Universal Robots PolyScope program: rtde_control_loop.urp

Program rtde_control_loop (installation=default directory=/programs createdIn=3.2.19275 lastSavedIn=5.13.0 robotSerialNumber=20225502595)
Calibrated DH parameters: a=[0.000032, -0.354602, -0.349314, -0.000114, 0.000079, 0]; d=[0.162572, 168.876417, -198.440969, 29.697991, 0.099792, 0.099551]; alpha=[1.570395, -0.001391, 0.006062, 1.570232, -1.569128, 0]; deltaTheta=[0, -0.584958, 0.110941, 0.474028, -0.000001, 0]
InitVariablesNode
BeforeStart
  setp := Joint_6_name
  Script: rtde_set_watchdog("input_int_register_0", 1, "PAUSE")
Robot Program (runOnlyOnce=false)
  Script: sync()
  MoveJ speed 60 deg/s, acceleration 80 deg/s^2 (useActiveTCP=true) feature=Base
    Waypoint Waypoint_1: TCP in base x=-26.855 y=-347.092 z=270.918 mm, rx=-0.0078 ry=3.1136 rz=-0.0162 rad; joints [-75.407, -74.048, -112.936, -82.13, 91.685, 14.557] deg; TCP offset x=0 y=50 z=155 mm, rx=0 ry=0 rz=0 rad
  If read_input_integer_register(1)≟1
    Script: write_output_integer_register(0, 0)
    MoveL speed 250 mm/s, acceleration 1200 mm/s^2 (useActiveTCP=true) feature=Base
      Waypoint Variable (Variable): variable=setp
    URCap qb Grasp (qbrobotics, qbrobotics®) dataModel(control_mode=deflection, grasp_command=78, grasp_threshold=100, grasp_velocity=100, grasp_stiffness=0)
    MoveJ speed 60 deg/s, acceleration 80 deg/s^2 (useActiveTCP=true) feature=Base
      Waypoint Waypoint_1: TCP in base x=-26.855 y=-347.092 z=270.918 mm, rx=-0.0078 ry=3.1136 rz=-0.0162 rad; joints [-75.407, -74.048, -112.936, -82.13, 91.685, 14.557] deg
      Waypoint Waypoint_2: TCP in base x=181.876 y=-239.045 z=110.303 mm, rx=-0.0609 ry=3.1315 rz=0.0832 rad; joints [-37.025, -75.759, -136.666, -59.157, 92.873, 51.044] deg
    URCap qb Grasp (qbrobotics, qbrobotics®) dataModel(control_mode=position, grasp_stiffness=50, grasp_command=43, grasp_threshold=100, grasp_velocity=100)
  Script: write_output_integer_register(0, 1)
  Wait Sleep waitTime=0.1
  Script: sync()
Thread Thread_1 (runOnlyOnce=false)
  setp := Joint_6_name
  Loop Forever
    tmp := p[0,0,0,0,0,0]
    Script: tmp[0] = read_input_float_register(0)
    Script: tmp[1] = read_input_float_register(1)
    Script: tmp[2] = read_input_float_register(2)
    Script: tmp[3] = read_input_float_register(3)
    Script: tmp[4] = read_input_float_register(4)
    Script: tmp[5] = read_input_float_register(5)
    If tmp != p[0,0,0,0,0,0]
      setp := tmp
    Script: sync()
